(*
    OBSOLETE. Test suite for FB_CheckPositionStateWrite, which is itself
    obsolete under the LCLS_Tc_Motion (ND) framework. See the obsolescence
    note in FB_CheckPositionStateWrite.TcPOU for the rationale. File kept
    on disk for history; excluded from Library.plcproj so it does not
    compile.
*)
FUNCTION_BLOCK FB_CheckPositionStateWriteTest EXTENDS FB_TestSuite
VAR
END_VAR


TestSaveCheck();

METHOD TestSaveCheck
VAR_INST
    astPositionState: ARRAY[1..GeneralConstants.MAX_STATES] OF ST_PositionState;
    fbCheckPositionStateWrite: FB_CheckPositionStateWrite;
END_VAR

TEST('TestSaveCheck');

fbCheckPositionStateWrite(
    astPositionState:=astPositionState,
    bCheck:=FALSE,
    bSave:=TRUE,
);
fbCheckPositionStateWrite(
    astPositionState:=astPositionState,
    bCheck:=TRUE,
    bSave:=FALSE,
);
AssertFalse(fbCheckPositionStateWrite.bHadWrite, 'Saw a write when there was no write');
astPositionState[1].fPosition := astPositionState[1].fPosition + 1;
fbCheckPositionStateWrite(
    astPositionState:=astPositionState,
    bCheck:=TRUE,
    bSave:=FALSE,
);
AssertTrue(fbCheckPositionStateWrite.bHadWrite, 'Did not detect position value changed');

TEST_FINISHED();
END_METHOD

END_FUNCTION_BLOCK

(* stored: Version 1.1.0.1
   POU FB_CheckPositionStateWriteTest: Id {b175a6be-c3c4-40f4-b64f-a3c7b0cdcfa8}, SpecialFunc None
   Method TestSaveCheck: Id {12a88bc9-b208-416d-8a25-c714576b382f} *)
